// TwinCAT 3 PLC project HMI_Background
// ProgramVersion: 3.1.4022.1
// libraries:
//   Tc2_Standard, * (Beckhoff Automation GmbH)
//   Tc2_System, * (Beckhoff Automation GmbH)
//   Tc3_Module, * (Beckhoff Automation GmbH)
// project tree:
//   GVLs/ GlobalVar.TcGVL, G_HMI_Communication.TcGVL, HMI_Variable.TcGVL
//   / PlcTask.TcTTO
//   POUs/ controller_p.TcPOU, Controller_PRG.TcPOU, cycl_change.TcPOU, MAIN.TcPOU, ArrayFiller_P.TcPOU
// real-time tasks:
//   TASK PlcTask: cycle T#4ms, priority 20, ADS port 350

CONFIGURATION HMI_Background
    RESOURCE PLC ON TwinCAT3
        TASK PlcTask(INTERVAL := T#4ms, PRIORITY := 20);
        PROGRAM MAIN WITH PlcTask : MAIN;
    END_RESOURCE
END_CONFIGURATION

// ---- GVLs/GlobalVar.TcGVL
{attribute 'qualified_only'}
VAR_GLOBAL
	G_GlobalArry01 : ARRAY [0..99] OF INT;
	G_GlobalArry02 : ARRAY [0..99] OF INT;
	G_Cycle: INT:=1;
	G_Cycle2: int:=1;		
END_VAR

// ---- GVLs/G_HMI_Communication.TcGVL
{attribute 'qualified_only'}
VAR_GLOBAL
	xControll: BOOL:= FALSE;
	xAutoMode: BOOL:= FALSE;
	xConfirmNotifi: BOOL:= FALSE;
	xLightGrid: BOOL:= TRUE;
	xEmSwitch: BOOL:= TRUE;
	xScrewDoor: BOOL:= TRUE;
	iOverAllSpeed: REAL:= 76.86;
	
	xAxisXpositive: BOOL:= FALSE;
	xAxisYpositive: BOOL:= FALSE;
	xAxisZpositive: BOOL:= FALSE;
	xAxisCpositive: BOOL:= FALSE;
	
	xAxisXnegative: BOOL:= FALSE;
	xAxisYnegative: BOOL:= FALSE;
	xAxisZnegative: BOOL:= FALSE;
	xAxisCnegative: BOOL:= FALSE;
	
	//----------------------------------
	iDepragStatus: INT:= 1;
	iDepragStep: INT:= 2;
	rDepragTorque: REAL:= 0.86;
	iDepragAngle: INT:= 56;
	iDepragProgramNR: INT:= 28;
	rDepragCycleTime: REAL:= 1.3;
	iErrorMessage: INT:= 0;
	
END_VAR

// ---- GVLs/HMI_Variable.TcGVL
{attribute 'qualified_only'}
VAR_GLOBAL
	in_speedstep: INT:= 1;
	in_speed: INT:= 5;
	in_maxcount: INT:= 100;
	in_increment: INT:= 1;	
	incerement: INT:= 1;
	b_IncrementNow: BOOL;
	//-----------------------------------
	b_Controll: BOOL:= FALSE;
	b_ModeSelect: BOOL:= FALSE;
	b_ConfirmNotifi: BOOL:= FALSE;
	b_ClearNotifi: Bool:= false;
	b_LightGrid: BOOL:= TRUE;
	b_EmSwitch: BOOL:= TRUE;
	b_ScrewDoor: BOOL:= TRUE;
	i_OverAllSpeed2: REAL:= 76.86;
	b_ManualMovementMode: BOOL:= TRUE;
	//----------------------------------
	i_DepragStatus: INT:= 1;
	i_DepragStep: INT:= 2;
	r_DepragTorque: REAL:= 0.86;
	i_DepragAngle: INT:= 56;
	i_DepragProgramNR: INT:= 28;
	r_DepragCycleTime: REAL:= 1.3;
	i_ErrorMessage: INT:= 0;
	//-----------------------------------
	t_temp: INT:= 0;
END_VAR

// ---- POUs/MAIN.TcPOU
PROGRAM MAIN
VAR
	in_speedstep: INT:= 1;
	in_speed: INT:= 5;
	in_maxcount: INT:= 100;
	in_increment: INT:= 1;	
	incerement: INT:= 1;
	b_IncrementNow: BOOL;
	//-----------------------------------
	b_Controll: BOOL:= FALSE;
	b_ModeSelect: BOOL:= FALSE;
	b_ConfirmNotifi: BOOL:= FALSE;
	b_LightGrid: BOOL:= TRUE;
	b_EmSwitch: BOOL:= TRUE;
	b_ScrewDoor: BOOL:= TRUE;
	i_OverAllSpeed: REAL:= 76.86;
	//----------------------------------
	i_DepragStatus: INT:= 1;
	i_DepragStep: INT:= 2;
	r_DepragTorque: REAL:= 0.86;
	i_DepragAngle: INT:= 56;
	i_DepragProgramNR: INT:= 28;
	r_DepragCycleTime: REAL:= 1.3;
	i_ErrorMessage: INT:= 0;
	//-----------------------------------
	t_temp: INT:= 0;
END_VAR

IF HMI_Variable.b_ConfirmNotifi  THEN
	HMI_Variable.b_ClearNotifi := TRUE;
	HMI_Variable.i_ErrorMessage:= 0;
END_IF

END_PROGRAM

// ---- POUs/controller_p.TcPOU
FUNCTION_BLOCK controller_p
VAR_INPUT
	b_start: BOOL;
	t_time: TIME;
END_VAR		
VAR_OUTPUT
	x_trigger: BOOL;
END_VAR
VAR
	fb_Pulse1: TP;
	fb_Pulse2: TP;
	fb_ftrig1: F_TRIG;
	fb_ftrig2: F_TRIG;
	b_StartTimer1: BOOL;
	b_StartTimer2: BOOL;
END_VAR

IF b_start THEN
	fb_Pulse1(IN:=b_StartTimer1,PT:=t_time);
	fb_Pulse2(IN:=b_StartTimer2,PT:=t_time);
	
	fb_ftrig1.CLK:= fb_Pulse1.Q;
	fb_ftrig2.CLK:= fb_Pulse2.Q;
	
	IF NOT fb_Pulse1.Q AND NOT fb_Pulse2.Q THEN
		b_StartTimer1:= TRUE;
		b_StartTimer2:= FALSE;
		
	ELSIF fb_ftrig1.Q THEN
		b_StartTimer1:= FALSE;
		b_StartTimer2:= TRUE;
		
	ELSIF fb_ftrig2.Q THEN
		b_StartTimer1:= TRUE;
		b_StartTimer2:= FALSE;
	END_IF
	
ELSE
	b_StartTimer1:= FALSE;
	b_StartTimer2:= FALSE;
	x_trigger:= FALSE;
END_IF

END_FUNCTION_BLOCK

// ---- POUs/Controller_PRG.TcPOU
PROGRAM Controller_PRG
VAR
END_VAR

END_PROGRAM

// ---- POUs/cycl_change.TcPOU
FUNCTION cycl_change : INT
VAR_INPUT
	i_cycle_int: INT;
	i_increment: INT;
END_VAR
VAR

END_VAR



i_cycle_int := i_cycle_int + i_increment;
cycl_change := i_cycle_int;

END_FUNCTION

// ---- POUs/ArrayFiller_P.TcPOU
FUNCTION ArrayFiller_P : ARRAY [0..99] OF INT
VAR_INPUT
END_VAR
VAR
	_TempArry : ARRAY [0..99] OF INT;
 	Index: INT;
END_VAR

FOR Index := 0 TO 99 DO
  _TempArry [Index] := 2500 + INDEX;
END_FOR
ArrayFiller_P := _TempArry;

END_FUNCTION
